(* PLC project BlogProject.project, CODESYS CODESYS V3.5 SP14 Patch 3 *)
(* stored: creationDateTime 2021-10-07T21:07:45.1828241, modificationDateTime 2021-10-07T20:40:20.1109198 *)

FUNCTION_BLOCK mcStopSystem IMPLEMENTS itfAction
  VAR_OUTPUT
    SystemStop : BOOL;
  END_VAR

            
          

METHOD getAction : BOOL
                  SystemStop:=TRUE;
StopCommand:=FALSE;
                
END_METHOD
END_FUNCTION_BLOCK
